FUNCTION_BLOCK LinearClearLinkMC EXTENDS ClearLinkMC IMPLEMENTS I_LinearEncodedDrive
VAR_INPUT
	sensorDefaultState : BOOL;
	
	homeAt0 : BOOL;
	allowDualSideTraverse : BOOL; //allows motion between home to retractLimit
END_VAR
VAR
	homePosition : LREAL;
	extendLimitPosition : LREAL;
	
	homingComplete : BOOL;
	
	home AT %I* : BOOL;
	extendLimit AT %I* : BOOL;
	retractLimit AT %I* : BOOL;
	
	step : Homing;
	calculation : (IDLE, EXTEND, RETRACT, CALCULATE, DONE);
END_VAR

SUPER^();

override();

PROPERTY AtExtendLimit : BOOL
GET
AtExtendLimit := extendLimit <> sensorDefaultState;
END_GET
END_PROPERTY

{attribute 'monitoring':='call'}
PROPERTY AtHome : BOOL
GET
AtHome := home <> sensorDefaultState;
END_GET
END_PROPERTY

PROPERTY AtRetractLimit : BOOL
GET
AtRetractLimit := retractLimit <> sensorDefaultState;
END_GET
END_PROPERTY

METHOD PRIVATE calculatePositions : BOOL
(*
THIS METHOD IS ONLY TO BE CALLED IF homeAt0 IS FALSE

not all drives have their home sensor at the 0 position
the purpose of this method is to calculate the home position, under the assumption that the extend limit sensor is 0

implementation:
	start from home
	reach the extend limit and set position to 0
	return to the home sensor and set the home position to the current position
*)
CASE calculation OF
	IDLE:
		calculation := EXTEND;
		
	EXTEND:		
		IF AtExtendLimit THEN
			
			IF homeAt0 THEN
				extendLimitPosition := CurrentPosition;
				calculation := RETRACT;
			
			ELSIF setPosition(newPosition := 0) THEN
				extendLimitPosition := 0;
				calculation := RETRACT;
			END_IF
		
		ELSE
			moveContinuous(newDirection := MC_Negative_Direction);
		END_IF
		
	RETRACT:
		IF AtHome THEN
			
			IF homeAt0 THEN
				homePosition := 0;
				calculation := DONE;
			
			ELSE
				homePosition := CurrentPosition;
				calculation := DONE;
			END_IF
		
		ELSE
			moveContinuous(newDirection := MC_Positive_Direction);
		END_IF
		
	DONE:
		calculation := 0;
		calculatePositions := TRUE;
		
END_CASE
END_METHOD

{attribute 'monitoring':='call'}
PROPERTY HomeSet : BOOL
GET
HomeSet := homingComplete;
END_GET
END_PROPERTY

METHOD homingSequence : BOOL
(*
homing sequence is different for linear motion devices with limit sensors
*)
CASE step OF
	Homing.IDLE:
		reset();
		IF bEnable THEN
			step := Homing.RETRY;
		END_IF
		
	Homing.START:
		IF AtHome THEN
			step := Homing.STOP;
			
		ELSIF AtRetractLimit THEN
			step := Homing.RETRY;
			
		ELSE
			moveContinuous(newDirection:= MC_Positive_Direction);
		END_IF
		
	Homing.RETRY:
		IF AtExtendLimit THEN
			step := Homing.START;
		ELSE
			moveContinuous(newDirection:= MC_Positive_Direction);
		END_IF
		
	Homing.STOP:
		IF stop() THEN
			step := Homing.SET;
		END_IF
		
	Homing.SET:
		IF calculatePositions() THEN
			step := Homing.DONE;
		END_IF
		
	Homing.DONE:
		homingComplete := TRUE;
		step := Homing.IDLE;
		
END_CASE
END_METHOD

METHOD PROTECTED override : BOOL
VAR_INPUT
END_VAR
IF AtHome AND NOT Active THEN
	IF homingDirectionOut THEN //homing is outwards
		position := maxPosition;
		pulsePosition := pulseCounter;
	ELSE
		position := minPosition;
		pulsePosition := 0;
	END_IF
	

ELSIF AtExtendLimit AND NOT Active THEN
	IF homingDirectionOut THEN //homing is outwards
		position := minPosition;
		pulsePosition := 0;
	ELSE
		position := maxPosition;
		pulsePosition := pulseCounter;
	END_IF
END_IF

IF
	(AtRetractLimit AND NOT A) OR
	(NOT allowDualSideTraverse AND AtHome AND A) OR
	(AtExtendLimit AND A)
THEN
	stop();
END_IF
(*
CASE mode OF		
	HOLD:
		//
	
	TARGET:
		IF
			(AtHome AND TargetPosition > CurrentPosition) OR
			(AtExtendLimit AND TargetPosition > CurrentPosition) OR
			(AtRetractLimit AND TargetPosition < CurrentPosition)
		THEN
			mode := HOLD;
		END_IF
		
	CONTINUOUS:
		IF
			(AtHome AND A) OR
			(AtExtendLimit AND A) OR
			(AtRetractLimit AND NOT A)
		THEN
			mode := HOLD;
		END_IF
		
	RESET_ERR:
		//
		
END_CASE
*)
END_METHOD

METHOD toHome : BOOL
VAR_INPUT
END_VAR
moveAbsolute(newTarget := homePosition);
END_METHOD

END_FUNCTION_BLOCK

(* stored: Version 1.1.0.1, ProductVersion 3.1.4024.11
   POU LinearClearLinkMC: Id {5cc69c24-a209-4ab4-827d-c3e832f18950}, SpecialFunc None
   Folder Properties: Id {a6689965-902c-4b2d-ac26-047bdef01e0c}
   Property AtExtendLimit: Id {1528a7d1-692e-4f26-bcbc-f2c7935a77e0}
   Get Get: Id {2d6acb00-d05a-4c9d-a7b4-a149a10d1124}
   Property AtHome: Id {cb359e28-f20d-4484-88d5-619a8ee99eab}
   Get Get: Id {03fbf48a-50db-4cd1-8ca7-a632d42ea4ab}
   Property AtRetractLimit: Id {aa495962-2e05-40e3-899e-34a650de2699}
   Get Get: Id {1264418a-2081-4312-8107-daa030ae7f6e}
   Method calculatePositions: Id {369fe372-e2d6-4f6c-8b9b-fc3030578aef}
   Property HomeSet: Id {098f2bde-4f8f-4326-9f57-7c66a1399c38}
   Get Get: Id {2b110dac-1b0f-41fe-a281-30a78b23ffd3}
   Method homingSequence: Id {0c6df03b-769b-4994-9517-30de0da8b72a}
   Method override: Id {0cbf85b0-6808-407c-97a7-52f87e0e0715}
   Method toHome: Id {de81265a-c215-460e-ab0a-8d476e0a3bcb} *)
